% RSLogix 500 project DIGITALCONTROLLOGIC_BAK001.RSS, saved by version 8.30.00.16 %
PROJECT "UNTITLED"    % processor: Bul.1763 MicroLogix 1100 Series A %

PROGRAM FILES
  LAD 2   3 rungs
  LAD 3 "I/O"  5 rungs  % Inupts and Outputs %
  LAD 4 "CONTROL"  9 rungs  % Control Logic %

DATA FILES
  O0 OUTPUT  4 elements
  I1 INPUT  6 elements
  S2 STATUS  66 elements
  B3 BINARY  1 elements
  T4 TIMER  1 elements
  C5 COUNTER  1 elements
  R6 CONTROL  1 elements
  N7 INTEGER  1 elements
  F8 FLOAT  1 elements

LADDER 2
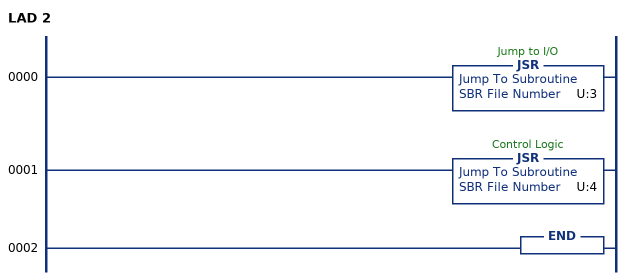
% Rung: 0 %  % edit flag set %
SOR JSR U:3 EOR
%   U:3  "Jump to I/O" %
% Rung: 1 %  % edit flag set %
SOR JSR U:4 EOR
%   U:4  "Control Logic" %
% Rung: 2 %
SOR END EOR

LADDER 3 "I/O"    % Inupts and Outputs %
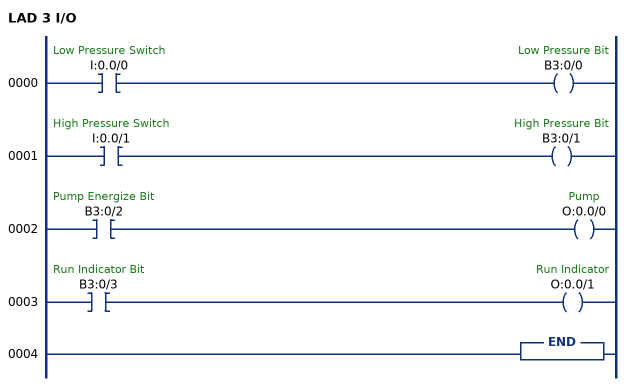
% Rung: 0 %  % edit flag set %
SOR XIC I:0.0/0 OTE B3:0/0 EOR
%   I:0.0/0  "Low Pressure Switch" %
%   B3:0/0  "Low Pressure Bit" %
% Rung: 1 %  % edit flag set %
SOR XIC I:0.0/1 OTE B3:0/1 EOR
%   I:0.0/1  "High Pressure Switch" %
%   B3:0/1  "High Pressure Bit" %
% Rung: 2 %  % edit flag set %
SOR XIC B3:0/2 OTE O:0.0/0 EOR
%   B3:0/2  "Pump Energize Bit" %
%   O:0.0/0  "Pump" %
% Rung: 3 %  % edit flag set %
SOR XIC B3:0/3 OTE O:0.0/1 EOR
%   B3:0/3  "Run Indicator Bit" %
%   O:0.0/1  "Run Indicator" %
% Rung: 4 %
SOR END EOR

LADDER 4 "CONTROL"    % Control Logic %
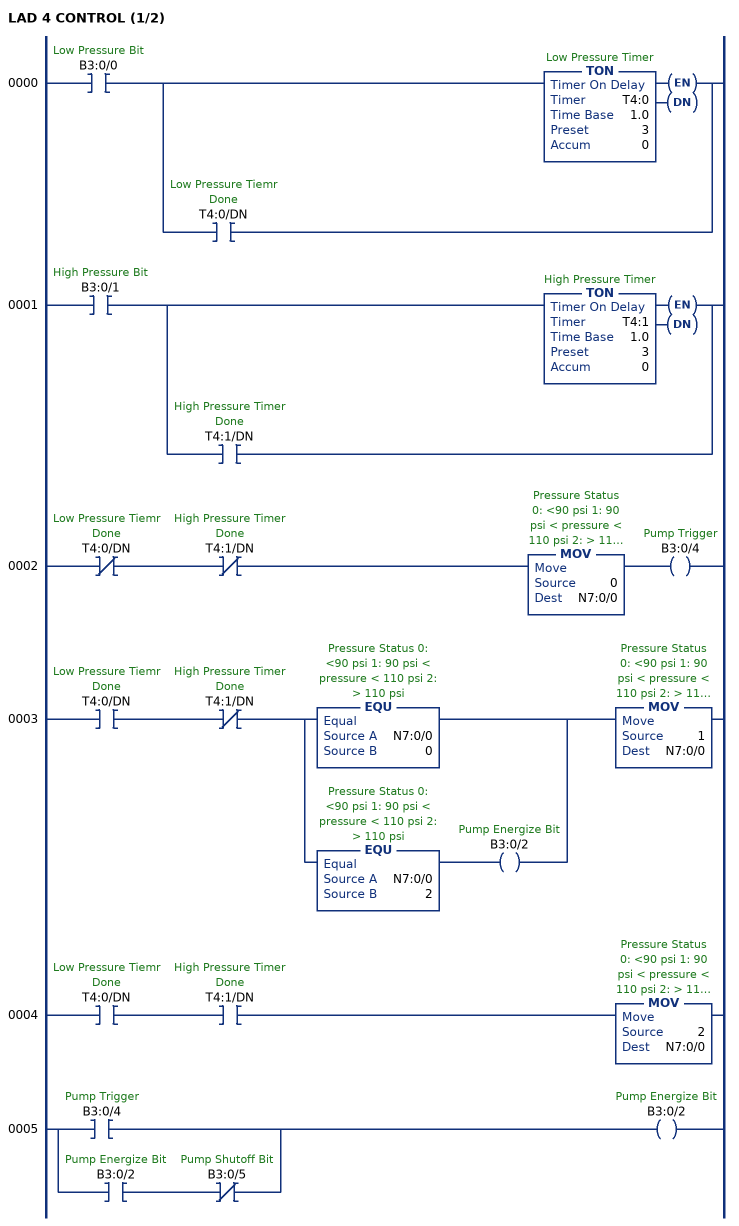
% Rung: 0 %  % edit flag set %
SOR XIC B3:0/0 BST TON T4:0 1.0 3 0 NXB XIC T4:0/DN BND EOR
%   B3:0/0  "Low Pressure Bit" %
%   T4:0  "Low Pressure Timer" %
%   T4:0/DN  "Low Pressure Tiemr Done" %
% Rung: 1 %  % edit flag set %
SOR XIC B3:0/1 BST TON T4:1 1.0 3 0 NXB XIC T4:1/DN BND EOR
%   B3:0/1  "High Pressure Bit" %
%   T4:1  "High Pressure Timer" %
%   T4:1/DN  "High Pressure Timer Done" %
% Rung: 2 %  % edit flag set %
SOR XIO T4:0/DN XIO T4:1/DN MOV 0 N7:0/0 OTE B3:0/4 EOR
%   T4:0/DN  "Low Pressure Tiemr Done" %
%   T4:1/DN  "High Pressure Timer Done" %
%   N7:0/0  "Pressure Status 0: <90 psi 1: 90 psi < pressure < 110 psi 2: > 110 psi" %
%   B3:0/4  "Pump Trigger" %
% Rung: 3 %  % edit flag set %
SOR XIC T4:0/DN XIO T4:1/DN BST EQU N7:0/0 0 NXB EQU N7:0/0 2 OTE B3:0/2 BND MOV 1 N7:0/0 EOR
%   T4:0/DN  "Low Pressure Tiemr Done" %
%   T4:1/DN  "High Pressure Timer Done" %
%   N7:0/0  "Pressure Status 0: <90 psi 1: 90 psi < pressure < 110 psi 2: > 110 psi" %
%   B3:0/2  "Pump Energize Bit" %
% Rung: 4 %  % edit flag set %
SOR XIC T4:0/DN XIC T4:1/DN MOV 2 N7:0/0 EOR
%   T4:0/DN  "Low Pressure Tiemr Done" %
%   T4:1/DN  "High Pressure Timer Done" %
%   N7:0/0  "Pressure Status 0: <90 psi 1: 90 psi < pressure < 110 psi 2: > 110 psi" %
% Rung: 5 %  % edit flag set %
SOR BST XIC B3:0/4 NXB XIC B3:0/2 XIO B3:0/5 BND OTE B3:0/2 EOR
%   B3:0/4  "Pump Trigger" %
%   B3:0/2  "Pump Energize Bit" %
%   B3:0/5  "Pump Shutoff Bit" %

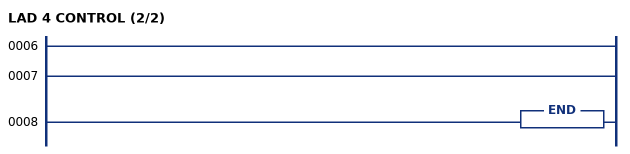
% Rung: 6 %  % edit flag set %
SOR EOR
% Rung: 7 %  % edit flag set %
SOR EOR
% Rung: 8 %
SOR END EOR
